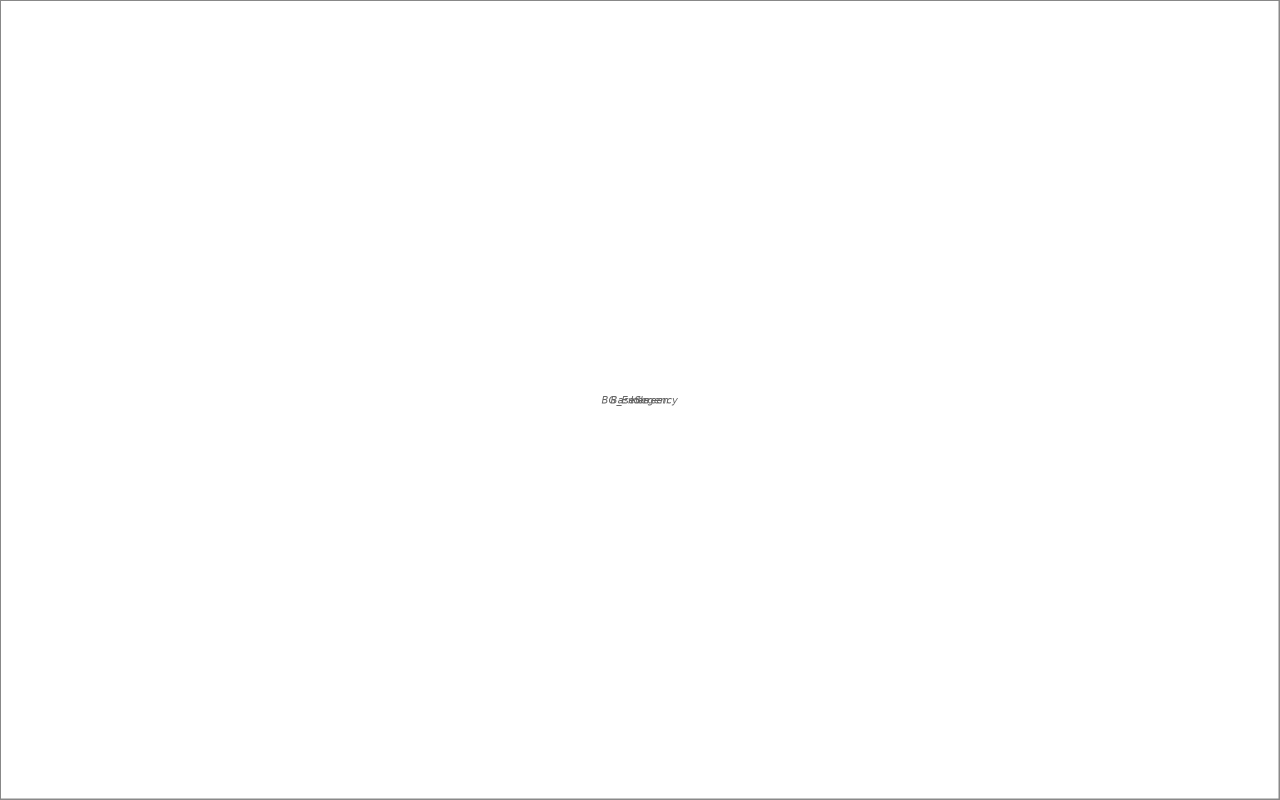
VISUALIZATION VISU_TEST_BASE  // 1280x800
    Frame (0,0 1280x800)
        shows BaseScreen()
    Frame (0,0 1280x800), frame switch variable: GVL_HMI.fbHMIControl.eShownScreen
        shows Idle()
        shows VISU_DummyState()
        shows Parameters()
        shows Manual()
        shows VISU_DummyState()
        shows VISU_DummyState()
        shows Log_()
    Frame (0,0 1280x800), invisible if: NOT GVL_HMI.fbHMIControl.bShowEmergencyOverlay
        shows BG_Emergency(sMessage := GVL_HMI.fbHMIControl.sEmergencyText)
END_VISUALIZATION

(* stored: Version 1.1.0.1, ProductVersion 3.1.4024.11
   Visu VISU_TEST_BASE: Id {be5d7be9-6163-4e15-836c-0969efcf4b70} *)
